// TIA Portal V17 export
// export: Created 2025-06-26T06:49:13.9283474Z, ExportSetting WithDefaults, DisplayName Totally Integrated Automation Portal, DisplayVersion V17 Update 8, DisplayName TIA Portal Openness, DisplayVersion V17 Update 8, DisplayName TIA Portal Version Control Interface, DisplayVersion V17, DisplayName STEP 7 Professional, DisplayVersion V17 Update 8, DisplayName STEP 7 Safety, DisplayVersion V17 Update 6, DisplayName WinCC Advanced, DisplayVersion V17 Update 8
FUNCTION_BLOCK "StateMachine"   // FB4, FBD
TITLE = Handling of machine states
{ S7_Optimized_Access := 'TRUE' }
VERSION : 0.1
// NB: the bit for each state stays high for one cycle after leaving the state. So when leaving State 2 for State 3, on the first cycle #StateChanges."2-zu-3_StateChange" will go high, setting the State 3 bit. But since the reset of State 2 is in an earlier network, this can't happen until the next cycle. So #StateChanges."2-zu-3_StateChange" has to stay high for the second cycle, when it causes State 2 RS to be reset. On the third cycle then also #StateChanges."2-zu-3_StateChange" is FALSE due to the State. This is subtle and tricky behaviour, not the best, rewrite this one day
// stored: AutoNumber true, IsIECCheckEnabled false, IsRetainMemResEnabled false, MemoryReserve 0, SetENOAutomatically false, UDAEnableTagReadback false
   VAR
      StateChanges : Struct
         "0-zu-1_StateChange" : Bool;
         "1-zu-2_StateChange" : Bool;
         "2-zu-3_StateChange" : Bool;
         "2-zu-7_StateChange" : Bool;
         "3-zu-2_StateChange" : Bool;
         "3-zu-4_StateChange" : Bool;
         "3-zu-7_StateChange" : Bool;
         "4-zu-2_StateChange" : Bool;
         "4-zu-5_StateChange" : Bool;
         "4-zu-7_StateChange" : Bool;
         "5-zu-2_StateChange" : Bool;
         "5-zu-6_StateChange" : Bool;
         "5-zu-7_StateChange" : Bool;
         "6-zu-2_StateChange" : Bool;
         "6-zu-7_StateChange" : Bool;
         "7-zu-1_StateChange" : Bool;
      END_STRUCT;
      Evaluate_DB : "Evaluate";
   END_VAR
   VAR_TEMP   // added for the SCL form of the ladder/FBD networks
      _w1 : Bool;
   END_VAR
BEGIN

REGION Network 1: Evaluate machine conditions
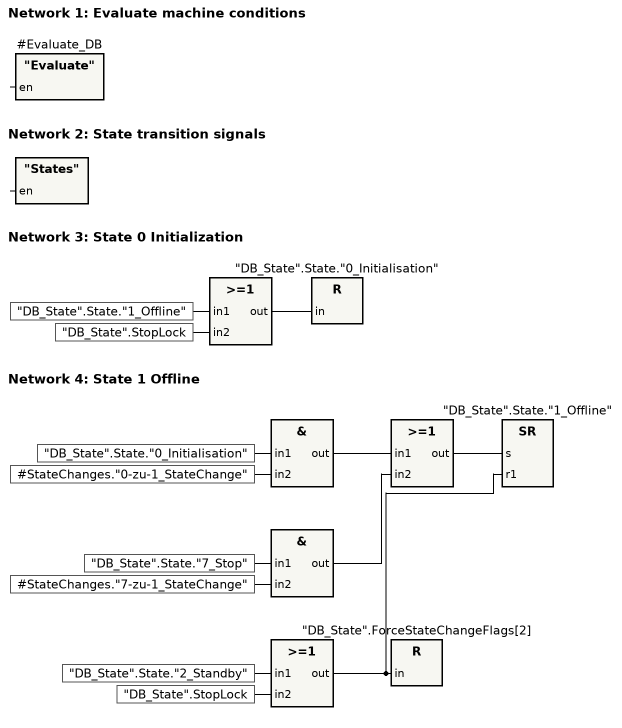
   #Evaluate_DB();   // "Evaluate"
END_REGION

REGION Network 2: State transition signals
   "States"();
END_REGION

REGION Network 3: State 0 Initialization
   // The "missing" SET logic is here:
   // Initialise (FB25) NW 2: "DB_StateMachine".State."0_Initialisation" := TRUE;
   IF "DB_State".State."1_Offline" OR "DB_State".StopLock THEN
       "DB_State".State."0_Initialisation" := FALSE;
   END_IF;
END_REGION

REGION Network 4: State 1 Offline
   #_w1 := "DB_State".State."2_Standby" OR "DB_State".StopLock;
   IF ("DB_State".State."0_Initialisation" AND #StateChanges."0-zu-1_StateChange") OR ("DB_State".State."7_Stop" AND #StateChanges."7-zu-1_StateChange") THEN
       "DB_State".State."1_Offline" := TRUE;   // SR flip-flop
   END_IF;
   IF #_w1 THEN
       "DB_State".State."1_Offline" := FALSE;
       "DB_State".ForceStateChangeFlags[2] := FALSE;
   END_IF;
END_REGION

REGION Network 5: State 2 Standby
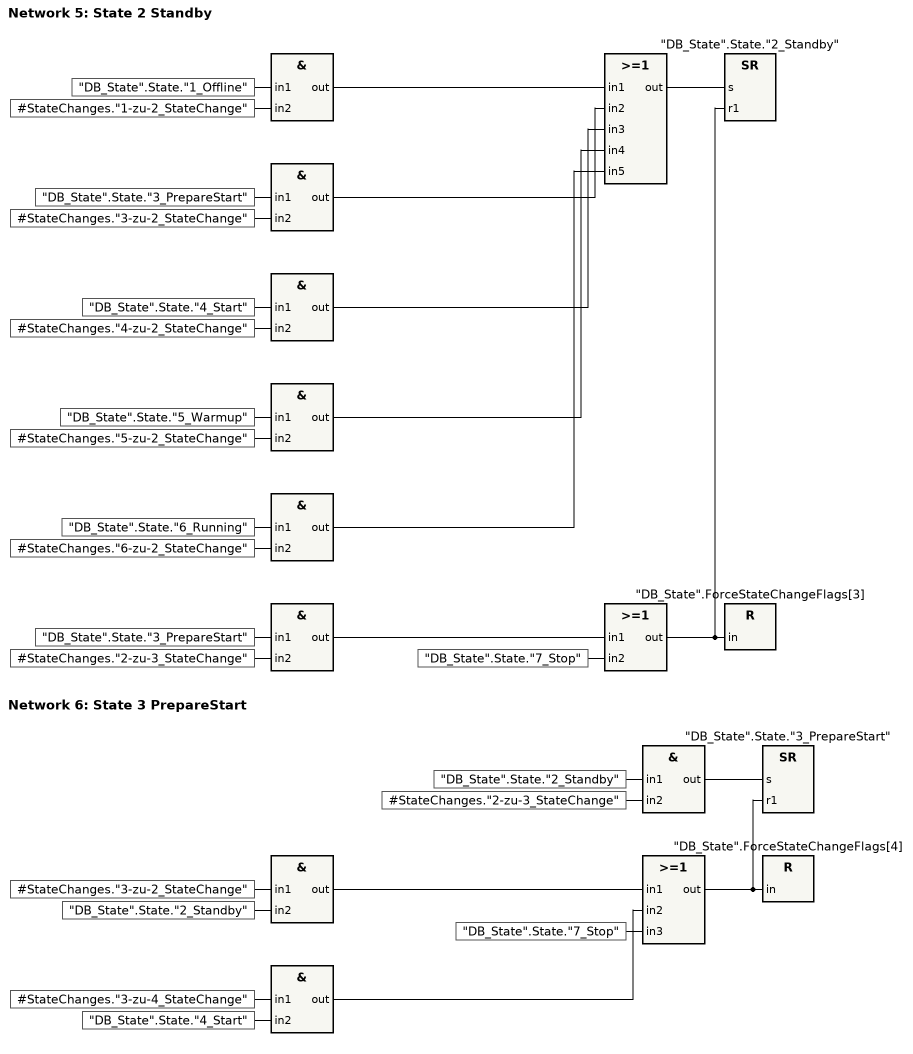
   #_w1 := ("DB_State".State."3_PrepareStart" AND #StateChanges."2-zu-3_StateChange") OR "DB_State".State."7_Stop";
   IF ("DB_State".State."1_Offline" AND #StateChanges."1-zu-2_StateChange") OR ("DB_State".State."3_PrepareStart" AND #StateChanges."3-zu-2_StateChange") OR ("DB_State".State."4_Start" AND #StateChanges."4-zu-2_StateChange") OR ("DB_State".State."5_Warmup" AND #StateChanges."5-zu-2_StateChange") OR ("DB_State".State."6_Running" AND #StateChanges."6-zu-2_StateChange") THEN
       "DB_State".State."2_Standby" := TRUE;   // SR flip-flop
   END_IF;
   IF #_w1 THEN
       "DB_State".State."2_Standby" := FALSE;
       "DB_State".ForceStateChangeFlags[3] := FALSE;
   END_IF;
END_REGION

REGION Network 6: State 3 PrepareStart
   #_w1 := (#StateChanges."3-zu-2_StateChange" AND "DB_State".State."2_Standby") OR (#StateChanges."3-zu-4_StateChange" AND "DB_State".State."4_Start") OR "DB_State".State."7_Stop";
   IF "DB_State".State."2_Standby" AND #StateChanges."2-zu-3_StateChange" THEN
       "DB_State".State."3_PrepareStart" := TRUE;   // SR flip-flop
   END_IF;
   IF #_w1 THEN
       "DB_State".State."3_PrepareStart" := FALSE;
       "DB_State".ForceStateChangeFlags[4] := FALSE;
   END_IF;
END_REGION

REGION Network 7: State 4 Start
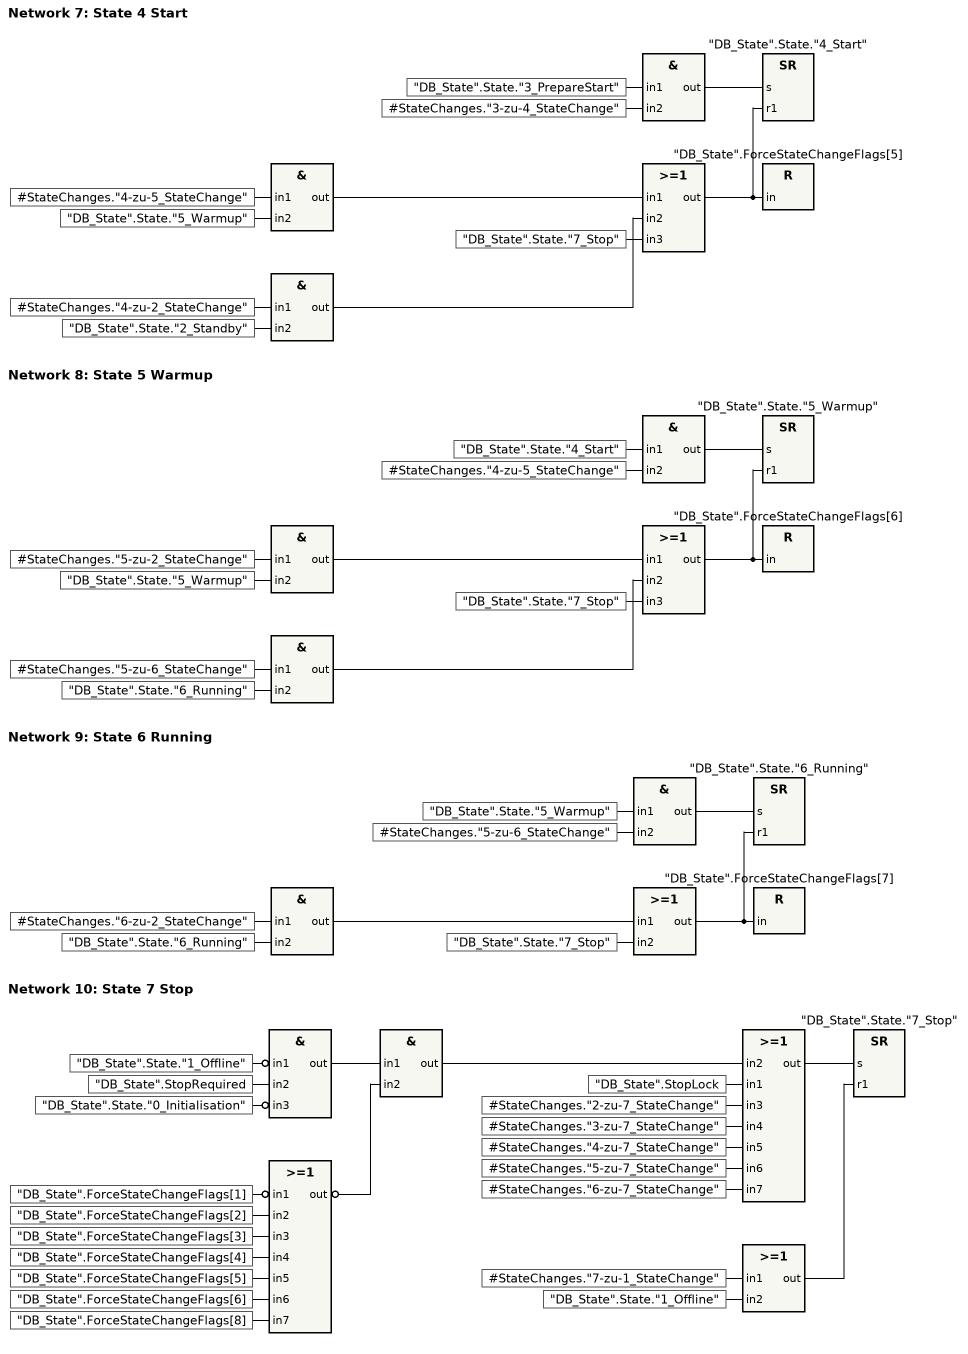
   #_w1 := (#StateChanges."4-zu-5_StateChange" AND "DB_State".State."5_Warmup") OR (#StateChanges."4-zu-2_StateChange" AND "DB_State".State."2_Standby") OR "DB_State".State."7_Stop";
   IF "DB_State".State."3_PrepareStart" AND #StateChanges."3-zu-4_StateChange" THEN
       "DB_State".State."4_Start" := TRUE;   // SR flip-flop
   END_IF;
   IF #_w1 THEN
       "DB_State".State."4_Start" := FALSE;
       "DB_State".ForceStateChangeFlags[5] := FALSE;
   END_IF;
END_REGION

REGION Network 8: State 5 Warmup
   #_w1 := (#StateChanges."5-zu-2_StateChange" AND "DB_State".State."5_Warmup") OR (#StateChanges."5-zu-6_StateChange" AND "DB_State".State."6_Running") OR "DB_State".State."7_Stop";
   IF "DB_State".State."4_Start" AND #StateChanges."4-zu-5_StateChange" THEN
       "DB_State".State."5_Warmup" := TRUE;   // SR flip-flop
   END_IF;
   IF #_w1 THEN
       "DB_State".State."5_Warmup" := FALSE;
       "DB_State".ForceStateChangeFlags[6] := FALSE;
   END_IF;
END_REGION

REGION Network 9: State 6 Running
   #_w1 := (#StateChanges."6-zu-2_StateChange" AND "DB_State".State."6_Running") OR "DB_State".State."7_Stop";
   IF "DB_State".State."5_Warmup" AND #StateChanges."5-zu-6_StateChange" THEN
       "DB_State".State."6_Running" := TRUE;   // SR flip-flop
   END_IF;
   IF #_w1 THEN
       "DB_State".State."6_Running" := FALSE;
       "DB_State".ForceStateChangeFlags[7] := FALSE;
   END_IF;
END_REGION

REGION Network 10: State 7 Stop
   IF (NOT "DB_State".State."1_Offline" AND "DB_State".StopRequired AND NOT "DB_State".State."0_Initialisation" AND NOT (NOT "DB_State".ForceStateChangeFlags[1] OR "DB_State".ForceStateChangeFlags[2] OR "DB_State".ForceStateChangeFlags[3] OR "DB_State".ForceStateChangeFlags[4] OR "DB_State".ForceStateChangeFlags[5] OR "DB_State".ForceStateChangeFlags[6] OR "DB_State".ForceStateChangeFlags[8])) OR "DB_State".StopLock OR #StateChanges."2-zu-7_StateChange" OR #StateChanges."3-zu-7_StateChange" OR #StateChanges."4-zu-7_StateChange" OR #StateChanges."5-zu-7_StateChange" OR #StateChanges."6-zu-7_StateChange" THEN
       "DB_State".State."7_Stop" := TRUE;   // SR flip-flop
   END_IF;
   IF #StateChanges."7-zu-1_StateChange" OR "DB_State".State."1_Offline" THEN
       "DB_State".State."7_Stop" := FALSE;
   END_IF;
END_REGION
END_FUNCTION_BLOCK
